FUNCTION_BLOCK E_MERGE (* Merge(OR)of multiple events *)
  (* Standard: 61499-2 *)
  (* Version 0.1, 2000-10-18, JHC, Rockwell Automation, XML version *)
  (* Version 0.0, 1998-11-19, JHC, Rockwell Automation, SRC version *)
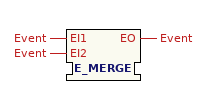
  EVENT_INPUT
    EI1; (* First input event *)
    EI2; (* Second input event *)
  END_EVENT
  EVENT_OUTPUT
    EO; (* Output Event *)
  END_EVENT
END_FUNCTION_BLOCK
